// TIA Portal V20 export
FUNCTION_BLOCK "LER_hipotHistory"   // FB36, LAD
// stored: Access Published, MemoryReserve 100, SetENOAutomatically false
   VAR_INPUT
      save : Bool;
      result : "LER_typePartData";
   END_VAR
   VAR_IN_OUT
      dataHistory : "LER_typeHipotHistory";
   END_VAR
   VAR
      statDeleteData { S7_SetPoint := 'True'} : "LER_typeHipotHistory";
      statTrigger : Array[0..9] of Bool;
      statTonTimer { S7_SetPoint := 'True'} : Array[0..99] of TON_TIME;
      statComplete { S7_SetPoint := 'True'} : Bool;
   END_VAR
   VAR_TEMP
      tempRetVal : Array[0..9] of Int;
   END_VAR
   VAR_TEMP   // added for the SCL form of the ladder/FBD networks
      _w1 : Bool;
   END_VAR
BEGIN

REGION Network 1
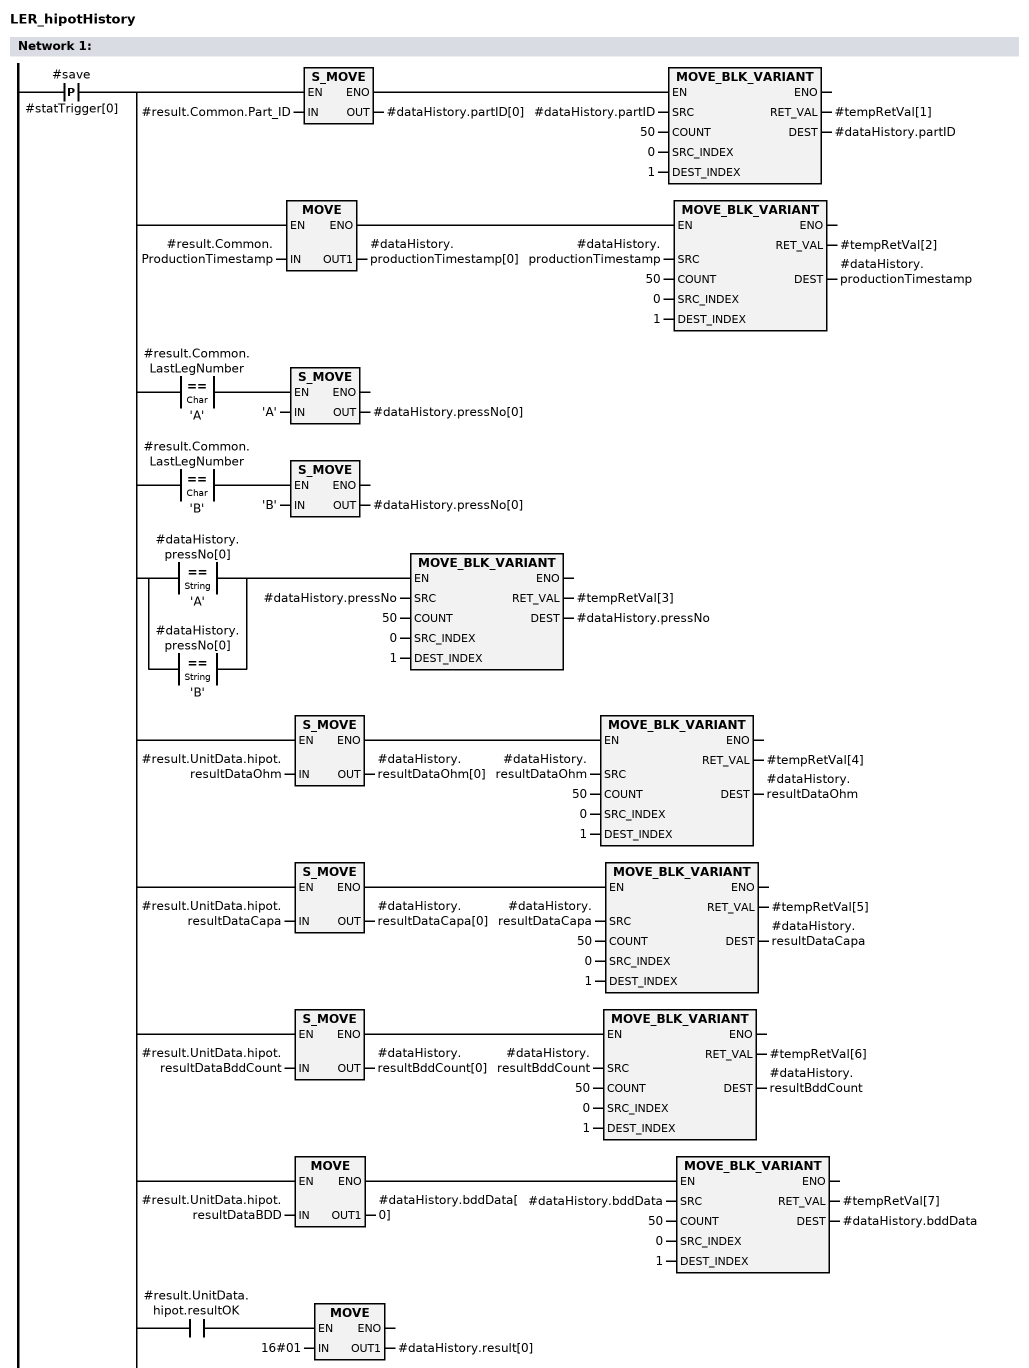
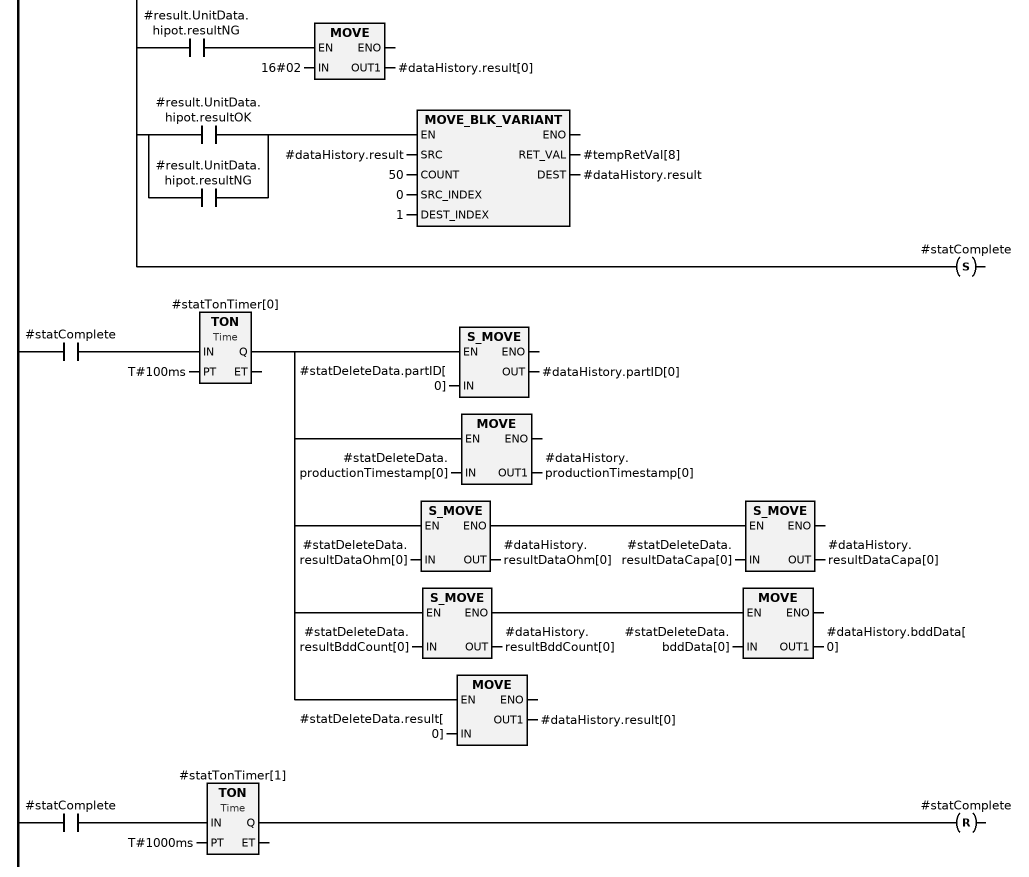
   RUNG wire#powerrail
      P_Contact(operand := #save, bit := #statTrigger[0])
      wire#w1
      S_Move(in := #result.Common.Part_ID, out => #dataHistory.partID[0])
      MOVE_BLK_VARIANT(SRC := #dataHistory.partID, COUNT := 50, SRC_INDEX := 0, DEST_INDEX := 1, Ret_Val => #tempRetVal[1], DEST => #dataHistory.partID)
   END_RUNG
   RUNG wire#w1
      Move(in := #result.Common.ProductionTimestamp, out1 => #dataHistory.productionTimestamp[0])
      MOVE_BLK_VARIANT(SRC := #dataHistory.productionTimestamp, COUNT := 50, SRC_INDEX := 0, DEST_INDEX := 1, Ret_Val => #tempRetVal[2], DEST => #dataHistory.productionTimestamp)
   END_RUNG
   RUNG wire#w1
      { S7_Templates := "SrcType := Char" } EQ_Contact(in1 := #result.Common.LastLegNumber, in2 := 'A')
      S_Move(in := 'A', out => #dataHistory.pressNo[0])
   END_RUNG
   RUNG wire#w1
      { S7_Templates := "SrcType := Char" } EQ_Contact(in1 := #result.Common.LastLegNumber, in2 := 'B')
      S_Move(in := 'B', out => #dataHistory.pressNo[0])
   END_RUNG
   RUNG wire#w1
      { S7_Templates := "SrcType := String" } EQ_Contact(in1 := #dataHistory.pressNo[0], in2 := 'A')
      wire#w2
      MOVE_BLK_VARIANT(SRC := #dataHistory.pressNo, COUNT := 50, SRC_INDEX := 0, DEST_INDEX := 1, Ret_Val => #tempRetVal[3], DEST => #dataHistory.pressNo)
   END_RUNG
   RUNG wire#w1
      { S7_Templates := "SrcType := String" } EQ_Contact(in1 := #dataHistory.pressNo[0], in2 := 'B')
   END_RUNG wire#w2
   RUNG wire#w1
      S_Move(in := #result.UnitData.hipot.resultDataOhm, out => #dataHistory.resultDataOhm[0])
      MOVE_BLK_VARIANT(SRC := #dataHistory.resultDataOhm, COUNT := 50, SRC_INDEX := 0, DEST_INDEX := 1, Ret_Val => #tempRetVal[4], DEST => #dataHistory.resultDataOhm)
   END_RUNG
   RUNG wire#w1
      S_Move(in := #result.UnitData.hipot.resultDataCapa, out => #dataHistory.resultDataCapa[0])
      MOVE_BLK_VARIANT(SRC := #dataHistory.resultDataCapa, COUNT := 50, SRC_INDEX := 0, DEST_INDEX := 1, Ret_Val => #tempRetVal[5], DEST => #dataHistory.resultDataCapa)
   END_RUNG
   RUNG wire#w1
      S_Move(in := #result.UnitData.hipot.resultDataBddCount, out => #dataHistory.resultBddCount[0])
      MOVE_BLK_VARIANT(SRC := #dataHistory.resultBddCount, COUNT := 50, SRC_INDEX := 0, DEST_INDEX := 1, Ret_Val => #tempRetVal[6], DEST => #dataHistory.resultBddCount)
   END_RUNG
   RUNG wire#w1
      Move(in := #result.UnitData.hipot.resultDataBDD, out1 => #dataHistory.bddData[0])
      MOVE_BLK_VARIANT(SRC := #dataHistory.bddData, COUNT := 50, SRC_INDEX := 0, DEST_INDEX := 1, Ret_Val => #tempRetVal[7], DEST => #dataHistory.bddData)
   END_RUNG
   RUNG wire#w1
      Contact( #result.UnitData.hipot.resultOK )
      Move(in := 16#01, out1 => #dataHistory.result[0])
   END_RUNG
   RUNG wire#w1
      Contact( #result.UnitData.hipot.resultNG )
      Move(in := 16#02, out1 => #dataHistory.result[0])
   END_RUNG
   RUNG wire#w1
      Contact( #result.UnitData.hipot.resultOK )
      wire#w3
      MOVE_BLK_VARIANT(SRC := #dataHistory.result, COUNT := 50, SRC_INDEX := 0, DEST_INDEX := 1, Ret_Val => #tempRetVal[8], DEST => #dataHistory.result)
   END_RUNG
   RUNG wire#w1
      Contact( #result.UnitData.hipot.resultNG )
   END_RUNG wire#w3
   RUNG wire#w1
      S_Coil( #statComplete )
   END_RUNG
   RUNG wire#powerrail
      Contact( #statComplete )
      { S7_Templates := "time_type := Time" } #statTonTimer[0].TON(pt := T#100ms, et =>)
      wire#w4
      S_Move(in := #statDeleteData.partID[0], out => #dataHistory.partID[0])
   END_RUNG
   RUNG wire#w4
      Move(in := #statDeleteData.productionTimestamp[0], out1 => #dataHistory.productionTimestamp[0])
   END_RUNG
   RUNG wire#w4
      S_Move(in := #statDeleteData.resultDataOhm[0], out => #dataHistory.resultDataOhm[0])
      S_Move(in := #statDeleteData.resultDataCapa[0], out => #dataHistory.resultDataCapa[0])
   END_RUNG
   RUNG wire#w4
      S_Move(in := #statDeleteData.resultBddCount[0], out => #dataHistory.resultBddCount[0])
      Move(in := #statDeleteData.bddData[0], out1 => #dataHistory.bddData[0])
   END_RUNG
   RUNG wire#w4
      Move(in := #statDeleteData.result[0], out1 => #dataHistory.result[0])
   END_RUNG
   RUNG wire#powerrail
      Contact( #statComplete )
      { S7_Templates := "time_type := Time" } #statTonTimer[1].TON(pt := T#1000ms, et =>)
      R_Coil( #statComplete )
   END_RUNG
   // the same network as SCL:
   #_w1 := #save AND NOT #statTrigger[0];   // rising edge of #save
   #statTrigger[0] := #save;
   IF #_w1 THEN
       #dataHistory.partID[0] := #result.Common.Part_ID;
       #tempRetVal[1] := MOVE_BLK_VARIANT(SRC := #dataHistory.partID,
                               COUNT := 50,
                               SRC_INDEX := 0,
                               DEST_INDEX := 1,
                               DEST => #dataHistory.partID);
       #dataHistory.productionTimestamp[0] := #result.Common.ProductionTimestamp;
       #tempRetVal[2] := MOVE_BLK_VARIANT(SRC := #dataHistory.productionTimestamp,
                               COUNT := 50,
                               SRC_INDEX := 0,
                               DEST_INDEX := 1,
                               DEST => #dataHistory.productionTimestamp);
   END_IF;
   IF #_w1 AND (#result.Common.LastLegNumber = 'A') THEN #dataHistory.pressNo[0] := 'A'; END_IF;
   IF #_w1 AND (#result.Common.LastLegNumber = 'B') THEN #dataHistory.pressNo[0] := 'B'; END_IF;
   IF #_w1 AND ((#dataHistory.pressNo[0] = 'A') OR (#dataHistory.pressNo[0] = 'B')) THEN
       #tempRetVal[3] := MOVE_BLK_VARIANT(SRC := #dataHistory.pressNo,
                               COUNT := 50,
                               SRC_INDEX := 0,
                               DEST_INDEX := 1,
                               DEST => #dataHistory.pressNo);
   END_IF;
   IF #_w1 THEN
       #dataHistory.resultDataOhm[0] := #result.UnitData.hipot.resultDataOhm;
       #tempRetVal[4] := MOVE_BLK_VARIANT(SRC := #dataHistory.resultDataOhm,
                               COUNT := 50,
                               SRC_INDEX := 0,
                               DEST_INDEX := 1,
                               DEST => #dataHistory.resultDataOhm);
       #dataHistory.resultDataCapa[0] := #result.UnitData.hipot.resultDataCapa;
       #tempRetVal[5] := MOVE_BLK_VARIANT(SRC := #dataHistory.resultDataCapa,
                               COUNT := 50,
                               SRC_INDEX := 0,
                               DEST_INDEX := 1,
                               DEST => #dataHistory.resultDataCapa);
       #dataHistory.resultBddCount[0] := #result.UnitData.hipot.resultDataBddCount;
       #tempRetVal[6] := MOVE_BLK_VARIANT(SRC := #dataHistory.resultBddCount,
                               COUNT := 50,
                               SRC_INDEX := 0,
                               DEST_INDEX := 1,
                               DEST => #dataHistory.resultBddCount);
       #dataHistory.bddData[0] := #result.UnitData.hipot.resultDataBDD;
       #tempRetVal[7] := MOVE_BLK_VARIANT(SRC := #dataHistory.bddData,
                               COUNT := 50,
                               SRC_INDEX := 0,
                               DEST_INDEX := 1,
                               DEST => #dataHistory.bddData);
   END_IF;
   IF #_w1 AND #result.UnitData.hipot.resultOK THEN #dataHistory.result[0] := 16#01; END_IF;
   IF #_w1 AND #result.UnitData.hipot.resultNG THEN #dataHistory.result[0] := 16#02; END_IF;
   IF #_w1 AND (#result.UnitData.hipot.resultOK OR #result.UnitData.hipot.resultNG) THEN
       #tempRetVal[8] := MOVE_BLK_VARIANT(SRC := #dataHistory.result,
                               COUNT := 50,
                               SRC_INDEX := 0,
                               DEST_INDEX := 1,
                               DEST => #dataHistory.result);
   END_IF;
   IF #_w1 THEN #statComplete := TRUE; END_IF;
   #statTonTimer[0].TON(IN := #statComplete, PT := T#100ms);
   IF #statTonTimer[0].Q THEN
       #dataHistory.partID[0] := #statDeleteData.partID[0];
       #dataHistory.productionTimestamp[0] := #statDeleteData.productionTimestamp[0];
       #dataHistory.resultDataOhm[0] := #statDeleteData.resultDataOhm[0];
       #dataHistory.resultDataCapa[0] := #statDeleteData.resultDataCapa[0];
       #dataHistory.resultBddCount[0] := #statDeleteData.resultBddCount[0];
       #dataHistory.bddData[0] := #statDeleteData.bddData[0];
       #dataHistory.result[0] := #statDeleteData.result[0];
   END_IF;
   #statTonTimer[1].TON(IN := #statComplete, PT := T#1000ms);
   IF #statTonTimer[1].Q THEN #statComplete := FALSE; END_IF;
END_REGION
END_FUNCTION_BLOCK
